// TwinCAT 3 PLC project PLC_Refrigirator_prj1
// ProgramVersion: 3.1.4023.0
// libraries:
//   Tc2_Standard, * (Beckhoff Automation GmbH)
//   Tc2_System, * (Beckhoff Automation GmbH)
//   Tc3_Module, * (Beckhoff Automation GmbH)
//   VisuDialogs, * (System)
//   VisuSymbols,3.5.10.0,System
// project tree:
//   / GlobalTextList.TcGTLO (not stored), PlcTask.TcTTO, Visualisierungsmanager.TcVMO (not stored)
//   GVLs/ GVL_Var.TcGVL (not stored)
//   POUs/ FB_Blinker.TcPOU, MAIN.TcPOU, Signals.TcPOU, Simulation.TcPOU (not stored)
//   VISUs/ Visualization.TcVIS (not stored)

CONFIGURATION PLC_Refrigirator_prj1
    RESOURCE PLC ON TwinCAT3
        TASK PlcTask(INTERVAL := T#10ms, PRIORITY := 20);
        PROGRAM MAIN WITH PlcTask : MAIN;
        PROGRAM Simulation WITH PlcTask : Simulation;
    END_RESOURCE
END_CONFIGURATION

// ---- POUs/MAIN.TcPOU
PROGRAM MAIN
VAR
	fHysteresis: REAL := 1;
	fbSR: SR;
END_VAR
VAR // added by the converter: edge detectors and wires of the graphical bodies
    _w1, _w2 : ANY;
END_VAR

fbSR(SET1 := _w1, RESET := GVL_Var.fTempActual < GVL_Var.fTempSet - fHysteresis); // SR
_w1 := GVL_Var.fTempActual > _w2;
_w2 := GVL_Var.fTempSet + fHysteresis;
GVL_Var.bCompressor := fbSR.Q1;
Signals();

END_PROGRAM

// ---- POUs/Signals.TcPOU
PROGRAM Signals
VAR
	fbTimer1: TON;
	fbTimer2: TON;
	FB_Blinker1: FB_Blinker;
END_VAR

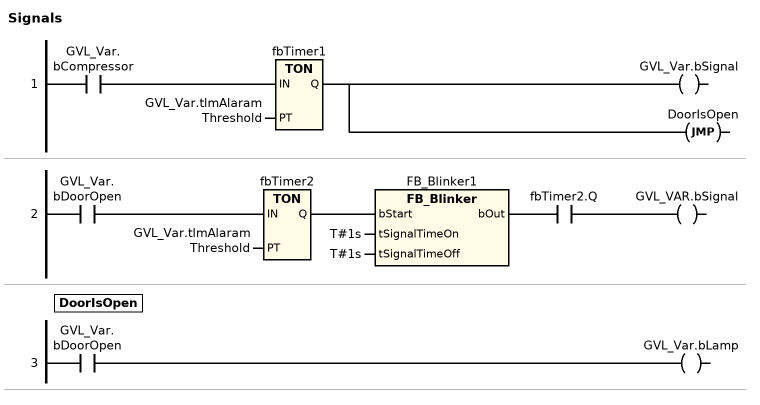
// NETWORK 1
fbTimer1(IN := GVL_Var.bCompressor, PT := GVL_Var.tlmAlaramThreshold); // TON
GVL_Var.bSignal := fbTimer1.Q;
IF fbTimer1.Q THEN JMP DoorIsOpen; END_IF

// NETWORK 2
fbTimer2(IN := GVL_Var.bDoorOpen, PT := GVL_Var.tlmAlaramThreshold); // TON
FB_Blinker1(bStart := fbTimer2.Q, tSignalTimeOn := T#1s, tSignalTimeOff := T#1s); // FB_Blinker
GVL_VAR.bSignal := FB_Blinker1.bOut AND fbTimer2.Q;

// NETWORK 3
DoorIsOpen:
GVL_Var.bLamp := GVL_Var.bDoorOpen;

END_PROGRAM

// ---- POUs/FB_Blinker.TcPOU
FUNCTION_BLOCK FB_Blinker
VAR_INPUT
	bStart: BOOL;
	tSignalTimeOn: TIME;
	tSignalTimeOff: TIME;
END_VAR
VAR_OUTPUT
	bOut: BOOL;
END_VAR
VAR
	fbTimerA: TON;
	fbTimerB: TON;
END_VAR

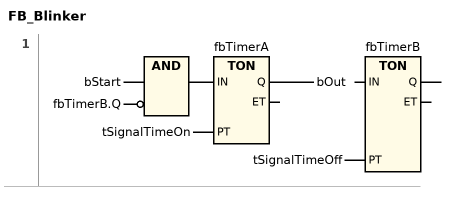
// NETWORK 1
fbTimerA(IN := bStart AND NOT fbTimerB.Q, PT := tSignalTimeOn); // TON
bOut := fbTimerA.Q;
fbTimerB(IN := fbTimerA.Q, PT := tSignalTimeOff); // TON

END_FUNCTION_BLOCK
